PROGRAM P_HTTP_Request
VAR
	DUT_Tls : ST_IotSocketTls;	
	fbIoTHTTP_Client: FB_IotHttpClient := (sHostName := 'api.openweathermap.org');
END_VAR

END_PROGRAM

(* stored: Version 1.1.0.1, ProductVersion 3.1.4024.12
   POU P_HTTP_Request: Id {90af155f-0f2d-4851-84f9-6a75f8fe52d5}, SpecialFunc None *)
